// Mitsubishi GX Works2 project: 타이머 문제3번풀이   PLC: Q02/Q02H

PROGRAM MAIN
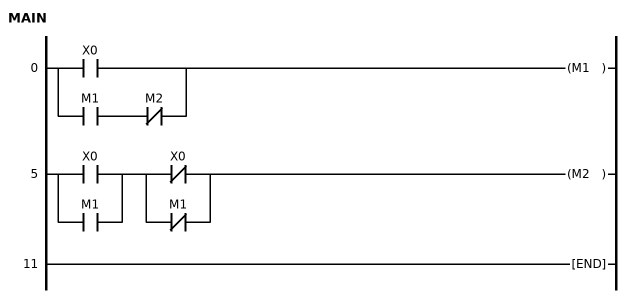
0     LD      X0
      LD      M1
      ANI     M2
      ORB
      OUT     M1
5     LD      X0
      OR      M1
      LDI     X0
      ORI     M1
      ANB
      OUT     M2
11    END
END_PROGRAM
